// TIA Portal V20 export
TYPE "PII - JN2200"
   STRUCT
      "Process Data Input - Angle Y / vibration acceleration Peak_max" : Int;
      "Process Data Input - Angle X / effective value of the vibration velocity" : Int;
      "Process Data Input - Diagnosis" : Byte;
      "Process Data Input - OUT1" : Bool;
      "Process Data Input - OUT2" : Bool;
      "Reserved Bit" : Bool;
      "Reserved Bit_1" : Bool;
      "Process Data Input - Vibration measurement" : Bool;
      "Process Data Input - Selftest running" : Bool;
      "Reserved Bit_2" : Bool;
      "Reserved Bit_3" : Bool;
   END_STRUCT;
END_TYPE
